FUNCTION_BLOCK EL2878
VAR
	{attribute addProperty Name "WcState"}
	_wcState : WcStateInputToggle;
	{attribute addProperty Name "Info data"}
	_infoData : InfoDataBase;
	_io : EL2878_Data;
END_VAR

PROPERTY IO : REFERENCE TO EL2878_Data
GET
IO REF= _io;
END_GET
END_PROPERTY

PROPERTY WcState : REFERENCE TO WcStateInputToggle
GET
WcState REF= _wcState;
END_GET
END_PROPERTY

END_FUNCTION_BLOCK

(* stored: Version 1.1.0.1, ProductVersion 3.1.4024.9
   POU EL2878: Id {ea797cfb-03ad-02d0-148d-8994e05511d3}, SpecialFunc None
   Property IO: Id {e2beb726-6e35-0db1-02ab-eccbb37f050b}
   Get Get: Id {5db7d3b3-152d-0e46-2aba-bc871d4f0b19}
   Property WcState: Id {3bcbd143-0380-073c-21d1-a81636d113f2}
   Get Get: Id {d02298a5-8fdd-07ca-1536-688a02e17ed1} *)
